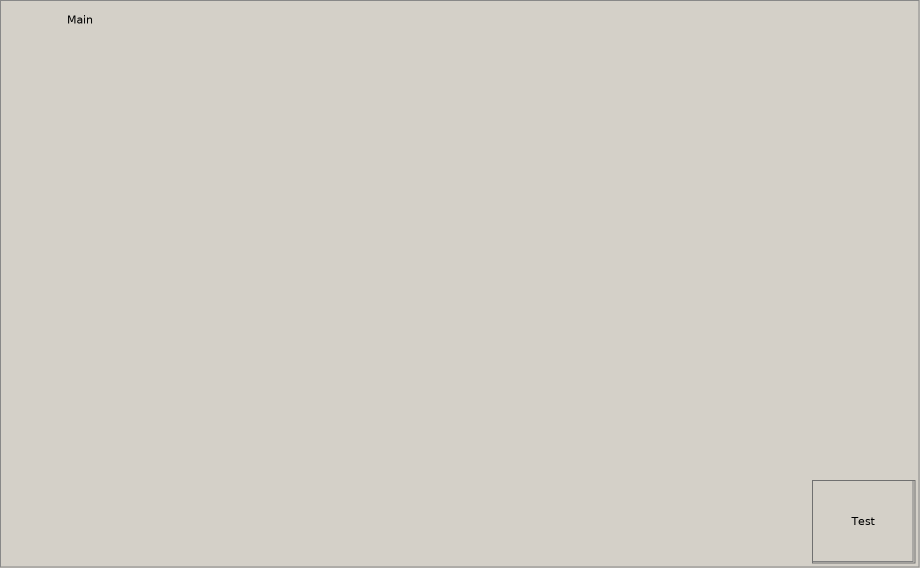
VISUALIZATION Main  // 920x568
    Label (5,5 150x30), "Main"
    Button (812,480 103x83), "Test", colour toggle: GVL_HMI.bTest
        toggle GVL_HMI.bTest
END_VISUALIZATION

(* stored: Version 1.1.0.1
   Visu Main: Id {f18f88ae-18d3-4de2-a8f3-ee47e837508b} *)
